# B&R Automation Studio project dbserv_0640 (part 4)

```c
/*=============================================================================
// Funktion: WorkEvent
//-----------------------------------------------------------------------------
// Zugriff auf das Prozessabbild.
// Input:	idBrServer: System-ID
// Return:	== 0 -> kein Fehler aufgetreten.
//			!= 0 -> Fehlerstatus der Funktion.
//=============================================================================*/

#ifdef FERTIG

UINT WorkEvent (void *idBrServer) {

	ACCESS_SERVER	*pAccessServer;
	ACCESS_UNIT		*pAccessUnit;
	ACCESS_TYPE		*pAccessType;
	ACCESS_POINT	*pAccessPoint;
	TYPE_DESC		*pTypeDesc;
	ITEM_DESC		*pItemDesc;

	ACCESS_ITEM_EVENT_LINK	*pAccessEventLinkItem;
	ACCESS_ITEM_EVENT_STATE	*pAccessEventItem;

	ACCESS_EVENT_PIPE	*pAccessEventPipe;
	EVENT_PIPE_HEADER	*pEventPipeHeader;
	EVENT_PIPE_DATA 	EventPipeData;
	USINT				*pEventPipeData, *pEventPipeTime;

	UDINT		lengthExtern, lengthPipeData, lengthTimeStamp;
	UINT		iPipeWrite, i;

	UINT		instance, unit, type, point, item;
	USINT		*pValue;
	UINT		lengthValue;
	USINT		eventtype;
	USINT		*pDataExtern;
	RTCtime_typ	RTCTime;

	if (idBrServer != NULL) {
		pAccessServer = (ACCESS_SERVER*)idBrServer;
		for (instance=0; instance<pAccessServer->countEventInstance; instance++) {
			for (unit=0; unit<pAccessServer->countUnit; unit++) {
				pAccessUnit = &pAccessServer->pAccessUnit[unit];
				if (pAccessUnit->pAccessType != NULL) {
					if (pAccessUnit->pUnitEventState[instance].countEvent > 0) {
						for (type=0; type<pAccessUnit->countType; type++) {
							pAccessType = &pAccessUnit->pAccessType[type];
							pTypeDesc = &pAccessServer->pAccessTypeDesc[type];
							if (pAccessType->pAccessPoint != NULL) {
								if (pAccessType->pTypeEventState[instance].countEvent > 0) {
									for (point=0; point<pAccessType->countPoint; point++) {
										pAccessPoint = &pAccessType->pAccessPoint[point];
										if (pAccessPoint->pAccessData != NULL) {
											if (pAccessPoint->pPointEventState[instance].countEvent > 0) {
												for (item=0; item<pTypeDesc->countItem ; item++) {
													pItemDesc = &pTypeDesc->pItemDesc[item];

													/* Event Datenbereich */
													pAccessEventItem = pAccessPoint->pAccessData + pAccessType->offiEvent + instance * pAccessType->leniEventNext + item * pAccessType->leniEventAlign;
													if (*pAccessEventItem == TRUE) {
														/* Link Datenbereich */
														pAccessEventLinkItem = pAccessPoint->pAccessData + pAccessType->offiEventlink + instance * pAccessType->leniEventlinkNext + item * pAccessType->leniEventlinkAlign;
														if (*pAccessEventLinkItem != cITEM_UNLINKED) {

															/* Daten wie für Funktions-Prototypen */
															pValue = pAccessPoint->pAccessData + pAccessType->offExtern + pItemDesc->offItem;
															lengthValue = pItemDesc->lenItem;
															eventtype = 0;
															pDataExtern = NULL;
															if (pAccessType->lenTime > 0) {
																memcpy(&RTCTime, pAccessPoint->pAccessData + pAccessType->offTime + item * pAccessType->lenTimeAlign, pAccessType->lenTime);
															}
															else {
																memset(&RTCTime, 0, sizeof(RTCTime));
															}

															/* SetEventItem */
															pAccessEventPipe = pAccessServer->pAccessEventPipe;
															lengthExtern = pItemDesc->lenItem;
															lengthTimeStamp = (*pAccessEventLinkItem == cITEM_LINKED_WITH_TIMESTAMP) ? sizeof(RTCtime_typ) : 0;
															pEventPipeHeader = (EVENT_PIPE_HEADER*)((USINT*)pAccessEventPipe[type].pEventPipeHeader + instance * pAccessEventPipe[type].length_pipe_next);
															lengthPipeData = (pValue != NULL) ? lengthValue : 0;
															if (pEventPipeHeader != NULL &&
																pEventPipeHeader->stateEvent.countEvent == 0 &&
																((pEventPipeHeader->iPipeWrite >= pEventPipeHeader->iPipeRead &&
																(UINT)(pEventPipeHeader->pipe_size - (pEventPipeHeader->iPipeWrite - pEventPipeHeader->iPipeRead)) > sizeof(EVENT_PIPE_DATA) + lengthTimeStamp + lengthPipeData) ||
																(pEventPipeHeader->iPipeWrite < pEventPipeHeader->iPipeRead &&
																(UINT)(pEventPipeHeader->iPipeRead - pEventPipeHeader->iPipeWrite) > sizeof(EVENT_PIPE_DATA) + lengthTimeStamp + lengthPipeData))) {

																if (pValue != NULL || pDataExtern != NULL) {
																	if ((pValue != NULL && lengthValue == lengthExtern) || pDataExtern != NULL) {
																		/* Eintrag in Event-Pipe */
																		iPipeWrite = pEventPipeHeader->iPipeWrite;

																		/* Header vorbesetzen */
																		EventPipeData.linkstate = *pAccessEventLinkItem;
																		EventPipeData.eventtype = eventtype;
																		EventPipeData.unit = unit;
																		EventPipeData.device = device;
																		EventPipeData.type = type;
																		EventPipeData.point= point;
																		EventPipeData.item = item;
																		EventPipeData.length = lengthValue;
																		EventPipeData.pData = pDataExtern;
																		pEventPipeData = (USINT*)&EventPipeData;
																		/* Header eintragen */
																		for (i=0; i<sizeof(EVENT_PIPE_DATA); i++) {
																			pEventPipeHeader->pPipeData[iPipeWrite++ % pEventPipeHeader->pipe_size] = pEventPipeData[i];
																		}
																		if (pValue != NULL) {
																			/* Daten eintragen */
																			for (i=0; i<lengthValue; i++) {
																				pEventPipeHeader->pPipeData[iPipeWrite++ % pEventPipeHeader->pipe_size] = pValue[i];
																			}
																		}
																		/* optional Zeitstempel eintragen */
																		if (lengthTimeStamp > 0) {
																			pEventPipeTime = (USINT*)&RTCTime;
																			for (i=0; i<lengthTimeStamp; i++) {
																				pEventPipeHeader->pPipeData[iPipeWrite++ % pEventPipeHeader->pipe_size] = pEventPipeTime[i];
																			}
																		}
																		/* Ereigniszeit aktualisieren */
																		if (pItemDesc->tsItem == TRUE) {
																			memcpy(pAccessPoint->pAccessData + pAccessType->offiTime + instance * pAccessType->leniTimeNext + item * pAccessType->leniTimeAlign, &RTCTime, pAccessType->leniTime);
																		}
																		pEventPipeHeader->iPipeWrite = (iPipeWrite % pEventPipeHeader->pipe_size); /* Index erst nach Zugriff updaten !!! */
																		pEventPipeHeader->pipe_level++; /* Füllstand erhöhen */

																	} /* ((pValue != NULL && lengthValue == lengthExtern) || pDataExtern != NULL) */
																	else {
																		return cEC_INVALID_LENGTH;
																	}
																} /* (pValue != NULL || pDataExtern != NULL) */
																else {
																	return cEC_INVALID_HANDLE;
																}
															}
														} /* (*pAccessEventLinkItem != cITEM_UNLINKED) */

														*pAccessEventItem = FALSE;
														pAccessPoint->pPointEventState[instance].countEvent--;
														pAccessType->pTypeEventState[instance].countEvent--;
														pAccessUnit->pUnitEventState[instance].countEvent--;

													} /* (*pAccessEventItem == TRUE) */
												} /* (item=0; item<pTypeDesc->countItem ; item++) */
											} /* (pAccessPoint->pPointEventState[instance] > 0) */
										} /* (pAccessPoint->pAccessData != NULL) */
									} /* (point=0; point<pAccessType->countPoint; point++) */
								} /* (pAccessType->pTypeEventState[instance].countEvent > 0) */
							} /* (pAccessType->pAccessPoint != NULL) */
						} /* (type=0; type<pAccessUnit->countType; type++) */
					} /* (pAccessUnit->pUnitEventState[instance].countEvent > 0) */
				} /* (pAccessUnit->pAccessType != NULL) */
			} /* (unit=0; unit<pAccessServer->countUnit; unit++) */
		} /* (instance=0; instance<pAccessServer->countEventInstance; instance++) */
		return cEC_OK;
	} /* (idBrServer != NULL) */
	else {
		return cEC_INVALID_SERVER;
	}
} /* WorkEvent */

/*UINT WorkEvent (void *idBrServer) {*/

	ACCESS_SERVER	*pAccessServer;
	ACCESS_UNIT		*pAccessUnit;
	ACCESS_TYPE		*pAccessType;
	ACCESS_POINT	*pAccessPoint;
	TYPE_DESC		*pTypeDesc;
	ITEM_DESC		*pItemDesc;
	ACCESS_ITEM_EVENT_LINK	*pAccessEventLinkItem;
	ACCESS_EVENT_PIPE		*pAccessEventPipe;
	EVENT_PIPE_HEADER		*pEventPipeHeader;

	UDINT					lengthExtern, lengthTimeStamp;
	UINT					i, instance, unit, device, type, point, iPipeWrite;

	EVENT_PIPE_DATA 		EventPipeData;
	USINT					*pEventPipeData, *pData, *pEventPipeTime;

	if (idBrServer != NULL) {
		pAccessServer = (ACCESS_SERVER*)idBrServer;
		for (instance=0; instance<pAccessServer->countEventInstance; instance++) {
			for (unit=0; unit<pAccessServer->countUnitNo; unit++) {
				pAccessUnit = &pAccessServer->pAccessUnit[unit];
				if (pAccessUnit->pAccessType != NULL) {
					if (pAccessServer->pUnitEventState[pAccessServer->countEventInstance * unit + instance].countEvent != 0) {
						for (device=0; device<pAccessUnit[unit].countDeviceNo; device++) {
							pAccessDevice = pAccessUnit[unit].pAccessDevice;
							if (device == pAccessDevice[device].device_no && pAccessDevice[device].pAccessType != NULL) {
								if (pAccessUnit[unit].pDeviceEventState[pAccessServer->countEventInstance * device + instance].countEvent != 0) {
									for (type=0; type<pAccessDevice[device].countType; type++) {
										if (pAccessDevice[device].pTypeEventState[pAccessServer->countEventInstance * type + instance].countEvent != 0) {

											pAccessType = pAccessDevice[device].pAccessType;
											pAccessEventPipe = pAccessServer->pAccessEventPipe;
											pEventPipeHeader = (EVENT_PIPE_HEADER*)((USINT*)pAccessEventPipe[type].pEventPipeHeader + instance * pAccessEventPipe[type].length_pipe_next);

											for (point=0; point<pAccessType[type].countPoint; point++) {

												pAccessEventLinkItem = pAccessType[type].pData_ieventlink + point * pAccessType[type].length_ieventlink_next;
												lengthExtern = pAccessEventPipe[type].TypeDefinition.length_extern;
												lengthTimeStamp = (pAccessEventLinkItem[instance] == cITEM_LINKED_WITH_TIMESTAMP) ? sizeof(RTCtime_typ) : 0;

												/* genügend Platz in der Event-Pipe ? */
												if (pEventPipeHeader != NULL &&
													pEventPipeHeader->stateEvent.countEvent != 0 &&
													((pEventPipeHeader->iPipeWrite >= pEventPipeHeader->iPipeRead &&
													(UINT)(pEventPipeHeader->pipe_size - (pEventPipeHeader->iPipeWrite - pEventPipeHeader->iPipeRead)) > sizeof(EVENT_PIPE_DATA) + lengthTimeStamp + lengthExtern) ||
													(pEventPipeHeader->iPipeWrite < pEventPipeHeader->iPipeRead &&
													(UINT)(pEventPipeHeader->iPipeRead - pEventPipeHeader->iPipeWrite) > sizeof(EVENT_PIPE_DATA) + lengthTimeStamp + lengthExtern))) {

													/* Event auf Datenpunkt vorhanden ? */
													if (*(UDINT*)(pAccessType[type].pData_ievent + point * pAccessType[type].length_ievent_next + instance * pAccessType[type].length_ievent_align) != 0 &&
														*(UDINT*)(pAccessType[type].pData_ievent + point * pAccessType[type].length_ievent_next + instance * pAccessType[type].length_ievent_align) == pEventPipeHeader->stateEvent.firstEvent) {

														/* Datenpunkt noch gelinkt ? */
														if (pAccessEventLinkItem[instance] != cITEM_UNLINKED) {

															/* Eintrag in Event-Pipe */
															iPipeWrite = pEventPipeHeader->iPipeWrite;

															/* Header eintragen */
															EventPipeData.linkstate = pAccessEventLinkItem[instance];
															EventPipeData.eventtype = 0;
															EventPipeData.unit = unit;
															EventPipeData.device = device;
															EventPipeData.type = type;
															EventPipeData.point= point;
															EventPipeData.item = 0;
															EventPipeData.length = lengthExtern;
															EventPipeData.pData = NULL;
															pEventPipeData = (USINT*)&EventPipeData;
															for (i=0; i<sizeof(EVENT_PIPE_DATA); i++) {
																pEventPipeHeader->pPipeData[iPipeWrite++ % pEventPipeHeader->pipe_size] = pEventPipeData[i];
															}

															/* Daten eintragen */
															pData = pAccessType[type].pData_extern + point * pAccessType[type].length_extern_align;
															for (i=0; i<lengthExtern; i++) {
																pEventPipeHeader->pPipeData[iPipeWrite++ % pEventPipeHeader->pipe_size] = pData[i];
															}
															pEventPipeHeader->iPipeWrite = (iPipeWrite % pEventPipeHeader->pipe_size); /* Index erst nach Zugriff updaten !!! */
															pEventPipeHeader->pipe_level++; /* Füllstand erhöhen */

															/* optional Zeitstempel eintragen */
															if (lengthTimeStamp > 0) {
																pEventPipeTime = pAccessType[type].pData_time + point * pAccessType[type].length_time_align;
																for (i=0; i<lengthTimeStamp; i++) {
																	pEventPipeHeader->pPipeData[iPipeWrite++ % pEventPipeHeader->pipe_size] = pEventPipeTime[i];
																}
															}
														} /* (pAccessItemLink[instance] != cITEM_UNLINKED) */

														/* Event auf Pipe-Typ austragen */
														pEventPipeHeader->stateEvent.firstEvent++;
														if (pEventPipeHeader->stateEvent.firstEvent > pEventPipeHeader->stateEvent.lastEvent) {
															pEventPipeHeader->stateEvent.firstEvent = 0;
															pEventPipeHeader->stateEvent.lastEvent = 0;
														}
														/* Event auf Punkt, Typ, Station, System austragen */
														*(UDINT*)(pAccessType[type].pData_ievent + point * pAccessType[type].length_ievent_next + instance * pAccessType[type].length_ievent_align) = 0;
														pEventPipeHeader->stateEvent.countEvent--;

														pAccessDevice[device].pTypeEventState[pAccessServer->countEventInstance * type + instance].countEvent--;
														pAccessUnit[unit].pDeviceEventState[pAccessServer->countEventInstance * device + instance].countEvent--;
														pAccessServer->pUnitEventState[pAccessServer->countEventInstance * unit + instance].countEvent--;

														/*if (pAccessServer->stateEvent[instance].countEvent == 0) {*/
															/* sicherheitshalber alle Pipe-Events bezüglich first/last austragen */
															/*for (m=0; m<pAccessServer->countType; m++) {
																pAccessEventPipe[m].stateEvent.firstEvent = 0;
																pAccessEventPipe[m].stateEvent.lastEvent = 0;
															}*/
														/*} (pAccessSystem->stateEvent.countEvent == 0) */
													} /* ... */
												} /* ... */
												else {
													break;
												}
											} /* (point=0; point<pAccessType[type].countPoint; point++) */
										} /* (pAccessDevice[device].pTypeEventState[pAccessServer->countEventInstance * type + instance].countEvent != 0) */
									} /* (type=0; type<pAccessDevice[device].countType; type++) */
								} /* (pAccessUnit[unit].pDeviceEventState[pAccessServer->countEventInstance * device + instance].countEvent != 0) */
							} /* (device == pAccessDevice[device].device_no && pAccessDevice[device].pAccessType != NULL) */
						} /* (device=0; device<pAccessUnit.countDeviceNo; device++) */
					} /* (pAccessServer->pUnitEventState[pAccessServer->countInstance * unit + instance].countEvent != 0) */
				} /* (unit == pAccessUnit[unit].unit_no && pAccessUnit[unit].pAccessDevice != NULL) */
			} /* (unit=0; unit<pAccessServer->countUnitNo; unit++) */
		} /* (instance=0; instance<pAccessServer->countEventInstance; instance++) */
		return cEC_OK;
	} /* (idBrServer != NULL) */
	else {
		return cEC_INVALID_SERVER;
	}
} /* work_event */
#endif

/*=============================================================================
// Funktion: LinkWriteInstance
//-----------------------------------------------------------------------------
// System mit allen zugehörigen Datenpunkten für die Ereignisbehandlung anmelden.
// Input:	idBrServer: System-ID
//			instance:	Instanz-Nummer
// Return:	== 0 -> kein Fehler aufgetreten.
//			!= 0 -> Fehlerstatus der Funktion.
//=============================================================================*/

UINT LinkWriteInstance (void *idBrServer, UINT instance) {

	ACCESS_SERVER	*pAccessServer;
	ACCESS_UNIT		*pAccessUnit;
	ACCESS_TYPE		*pAccessType;
	ACCESS_POINT	*pAccessPoint;
	TYPE_DESC		*pTypeDesc;
	ACCESS_ITEM_WRITE_LINK	*pAccessWriteLinkItem;

	unsigned short	unit, type, point, item;

	if (idBrServer != NULL) {
		pAccessServer = (ACCESS_SERVER*)idBrServer;
		if (instance < pAccessServer->countWriteInstance) {
			for (unit=0; unit<pAccessServer->countUnit; unit++) {
				pAccessUnit = &pAccessServer->pAccessUnit[unit];
				if (pAccessUnit->pAccessType != NULL) {
					for (type=0; type<pAccessUnit->countType; type++) {
						pAccessType = &pAccessUnit->pAccessType[type];
						pTypeDesc = &pAccessServer->pAccessTypeDesc[type];
						if (pAccessType->pAccessPoint != NULL) {
							for (point=0; point<pAccessType->countPoint; point++) {
								pAccessPoint = &pAccessType->pAccessPoint[point];
								if (pAccessPoint->pAccessData != NULL) {
									for (item=0; item<pTypeDesc->countItem ; item++) {
										/* Link Datenbereich */
										pAccessWriteLinkItem = pAccessPoint->pAccessData + pAccessType->offWritelink + item * pAccessType->lenWritelinkAlign;
										if (*pAccessWriteLinkItem == 0) {
											*pAccessWriteLinkItem = instance + 1;
										}
									} /* (item = 0; item<pTypeDesc->countItem ; item++) */
								} /* (pAccessPoint->pAccessData != NULL) */
							} /* (point=0; point<pAccessType->countPoint; point++) */
						} /* (pAccessType->pAccessPoint != NULL) */
					} /* (type=0; type<pAccessUnit->countType; type++) */
				} /* (pAccessUnit->pAccessType != NULL) */
			} /* (unit=0; unit<pAccessServer->countUnit; unit++) */
			return cEC_OK;
		} /* (instance < pAccessSystem->countWriteInstance) */
		else {
			return cEC_INVALID_INSTANCE;
		}
	} /* (idBrServer != NULL) */
	else {
		return cEC_INVALID_SERVER;
	}
} /* LinkWriteInstance */

/*=============================================================================
// Funktion: UnlinkWriteInstance
//-----------------------------------------------------------------------------
// System mit allen zugehörigen Datenpunkten für die Ereignisbehandlung anmelden.
// Input:	idBrServer: System-ID
//			instance:	Instanz-Nummer
// Return:	== 0 -> kein Fehler aufgetreten.
//			!= 0 -> Fehlerstatus der Funktion.
//=============================================================================*/

UINT UnlinkWriteInstance (void *idBrServer, UINT instance) {

	ACCESS_SERVER	*pAccessServer;
	ACCESS_UNIT		*pAccessUnit;
	ACCESS_TYPE		*pAccessType;
	ACCESS_POINT	*pAccessPoint;
	TYPE_DESC		*pTypeDesc;
	ACCESS_ITEM_WRITE_LINK	*pAccessWriteLinkItem;

	unsigned short	unit, type, point, item;

	if (idBrServer != NULL) {
		pAccessServer = (ACCESS_SERVER*)idBrServer;
		if (instance < pAccessServer->countWriteInstance) {
			for (unit=0; unit<pAccessServer->countUnit; unit++) {
				pAccessUnit = &pAccessServer->pAccessUnit[unit];
				if (pAccessUnit->pAccessType != NULL) {
					for (type=0; type<pAccessUnit->countType; type++) {
						pAccessType = &pAccessUnit->pAccessType[type];
						pTypeDesc = &pAccessServer->pAccessTypeDesc[type];
						if (pAccessType->pAccessPoint != NULL) {
							for (point=0; point<pAccessType->countPoint; point++) {
								pAccessPoint = &pAccessType->pAccessPoint[point];
								if (pAccessPoint->pAccessData != NULL) {
									for (item=0; item<pTypeDesc->countItem ; item++) {
										/* Unlink Datenbereich */
										pAccessWriteLinkItem = pAccessPoint->pAccessData + pAccessType->offWritelink + item * pAccessType->lenWritelinkAlign;
										if (*pAccessWriteLinkItem > 0) {
											*pAccessWriteLinkItem = 0;
										}
									} /* (item = 0; item<pTypeDesc->countItem ; item++) */
								} /* (pAccessPoint->pAccessData != NULL) */
							} /* (point=0; point<pAccessType->countPoint; point++) */
						} /* (pAccessType->pAccessPoint != NULL) */
					} /* (type=0; type<pAccessUnit->countType; type++) */
				} /* (pAccessUnit->pAccessType != NULL) */
			} /* (unit=0; unit<pAccessServer->countUnit; unit++) */
			return cEC_OK;
		} /* (instance < pAccessSystem->countWriteInstance) */
		else {
			return cEC_INVALID_INSTANCE;
		}
	} /* (idBrServer != NULL) */
	else {
		return cEC_INVALID_SERVER;
	}
} /* UnlinkWriteInstance */

/*=============================================================================
// Funktion: LinkWriteItem
//-----------------------------------------------------------------------------
// Datenpunkt für Ereignisbehandlung anmelden.
// Input:	idBrServer: System-ID
//			instance:	Instanz-Nummer
//			unit:		Anlagen-Nummer
//			device:		Gerät-Nummer
//			type:		Datentyp-Nummer
//			point:		Datenpunkt-Nummer
//			item:		Strukturelement-Nummer
// Return:	== 0 -> kein Fehler aufgetreten.
//			!= 0 -> Fehlerstatus der Funktion.
//=============================================================================*/

UINT LinkWriteItem (void *idBrServer, UINT instance,
					UINT unit, UINT device, UINT type, UINT point, UINT item,
					UDINT handle) {

	ACCESS_SERVER	*pAccessServer;
	ACCESS_UNIT		*pAccessUnit;
	ACCESS_TYPE		*pAccessType;
	ACCESS_POINT	*pAccessPoint;
	TYPE_DESC		*pTypeDesc;
	ITEM_DESC		*pItemDesc;
	ACCESS_ITEM_WRITE_LINK		*pAccessWriteLinkItem;
	ACCESS_ITEM_WRITE_HANDLE	*pAccessWriteHandleItem;

	if (idBrServer != NULL) {
		pAccessServer = (ACCESS_SERVER*)idBrServer;
		if (instance < pAccessServer->countWriteInstance) {
			if (unit < pAccessServer->countUnit && pAccessServer->pAccessUnit[unit].pAccessType != NULL) {
				pAccessUnit = &pAccessServer->pAccessUnit[unit];
				if (device == pAccessServer->noDevice) {
					if (type < pAccessUnit->countType && pAccessUnit->pAccessType[type].pAccessPoint != NULL) {
						pAccessType = &pAccessUnit->pAccessType[type];
						pTypeDesc = &pAccessServer->pAccessTypeDesc[type];
						if (point < pAccessType->countPoint && pAccessType->pAccessPoint[point].pAccessData != NULL) {
							pAccessPoint = &pAccessType->pAccessPoint[point];
							if (item < pTypeDesc->countItem) {
								pItemDesc = &pTypeDesc->pItemDesc[item];

								/* Link Datenbereich */
								pAccessWriteLinkItem = pAccessPoint->pAccessData + pAccessType->offWritelink + item * pAccessType->lenWritelinkAlign;
								pAccessWriteHandleItem = (ACCESS_ITEM_WRITE_HANDLE*)(pAccessPoint->pAccessData + pAccessType->offWritehandle + item * pAccessType->lenWritehandleAlign);
								if (*pAccessWriteLinkItem == 0) {
									*pAccessWriteLinkItem = instance + 1;
									*pAccessWriteHandleItem = handle;
									return cEC_OK;
								}
								else {
									return cEC_ITEM_ALREADY_LINKED;
								}

							} /* (item < pTypeDesc->countItem) */
							else {
								return cEC_INVALID_ITEM;
							}
						} /* (point < pAccessType->countPoint && pAccessType->pAccessPoint[point].pAccessData != NULL) */
						else {
							return cEC_INVALID_POINT;
						}
					} /* (type < pAccessUnit->countType && pAccessUnit->pAccessType[type].pAccessPoint != NULL) */
					else {
						return cEC_INVALID_TYPE;
					}
				} /* (device == pAccessServer->noDevice) */
				else {
					return cEC_INVALID_DEVICE;
				}
			} /* (unit < pAccessServer->countUnit) */
			else {
				return cEC_INVALID_UNIT;
			}
		} /* (instance < pAccessSystem->countWriteInstance) */
		else {
			return cEC_INVALID_INSTANCE;
		}
	} /* (idBrServer != NULL) */
	else {
		return cEC_INVALID_SERVER;
	}
} /* LinkWriteItem */

/*=============================================================================
// Funktion: UnlinkWriteItem
//-----------------------------------------------------------------------------
// Datenpunkt für Ereignisbehnadlung abmelden.
// Input:	idBrServer: System-ID
//			instance:	Instanz-Nummer
//			unit:		Anlagen-Nummer
//			device:		Gerät-Nummer
//			type:		Datentyp-Nummer
//			point:		Datenpunkt-Nummer
//			item:		Strukturelement-Nummer
// Return:	== 0 -> kein Fehler aufgetreten.
//			!= 0 -> Fehlerstatus der Funktion.
//=============================================================================*/

UINT UnlinkWriteItem (void *idBrServer, UINT instance,
						UINT unit, UINT device, UINT type, UINT point, UINT item) {

	ACCESS_SERVER	*pAccessServer;
	ACCESS_UNIT		*pAccessUnit;
	ACCESS_TYPE		*pAccessType;
	ACCESS_POINT	*pAccessPoint;
	TYPE_DESC		*pTypeDesc;
	ITEM_DESC		*pItemDesc;
	ACCESS_ITEM_WRITE_LINK		*pAccessWriteLinkItem;
	ACCESS_ITEM_WRITE_HANDLE	*pAccessWriteHandleItem;

	if (idBrServer != NULL) {
		pAccessServer = (ACCESS_SERVER*)idBrServer;
		if (instance < pAccessServer->countWriteInstance) {
			if (unit < pAccessServer->countUnit && pAccessServer->pAccessUnit[unit].pAccessType != NULL) {
				pAccessUnit = &pAccessServer->pAccessUnit[unit];
				if (device == pAccessServer->noDevice) {
					if (type < pAccessUnit->countType && pAccessUnit->pAccessType[type].pAccessPoint != NULL) {
						pAccessType = &pAccessUnit->pAccessType[type];
						pTypeDesc = &pAccessServer->pAccessTypeDesc[type];
						if (point < pAccessType->countPoint && pAccessType->pAccessPoint[point].pAccessData != NULL) {
							pAccessPoint = &pAccessType->pAccessPoint[point];
							if (item < pTypeDesc->countItem) {
								pItemDesc = &pTypeDesc->pItemDesc[item];

								/* Unlink Datenbereich */
								pAccessWriteLinkItem = pAccessPoint->pAccessData + pAccessType->offWritelink + item * pAccessType->lenWritelinkAlign;
								pAccessWriteHandleItem = (ACCESS_ITEM_WRITE_HANDLE*)(pAccessPoint->pAccessData + pAccessType->offWritehandle + item * pAccessType->lenWritehandleAlign);
								if (*pAccessWriteLinkItem > 0) {
									*pAccessWriteLinkItem = 0;
									*pAccessWriteHandleItem = 0;
									return cEC_OK;
								}
								else {
									return cEC_ITEM_ALREADY_UNLINKED;
								}

							} /* (item < pTypeDesc->countItem) */
							else {
								return cEC_INVALID_ITEM;
							}
						} /* (point < pAccessType->countPoint && pAccessType->pAccessPoint[point].pAccessData != NULL) */
						else {
							return cEC_INVALID_POINT;
						}
					} /* (type < pAccessUnit->countType && pAccessUnit->pAccessType[type].pAccessPoint != NULL) */
					else {
						return cEC_INVALID_TYPE;
					}
				} /* (device == pAccessServer->noDevice) */
				else {
					return cEC_INVALID_DEVICE;
				}
			} /* (unit < pAccessServer->countUnit && pAccessServer->pAccessUnit[unit].pAccessType != NULL) */
			else {
				return cEC_INVALID_UNIT;
			}
		} /* (instance < pAccessSystem->countWriteInstance) */
		else {
			return cEC_INVALID_INSTANCE;
		}
	} /* (idBrServer != NULL) */
	else {
		return cEC_INVALID_SERVER;
	}
} /* UnlinkWriteItem */

/*=============================================================================
// Funktion: SetWriteItem
//-----------------------------------------------------------------------------
// Zugriff auf das Prozessabbild.
// Input:	idBrServer: System-ID
//			system:		Anlagen-Nummer
//			station:	Stations-Nummer
//			type:		Datentyp-Nummer
//			point:		Datenpunkt-Nummer
//			ppData_extern:	Zeiger auf externen Datenbereich (Rückgabewert)
//			plength_extern:	Länge des externen Datenbereichs (Rückgabewert)
//			ppData_intern:	Zeiger auf internen Datenbereich (Rückgabewert)
//			plength_intern:	Länge des internen Datenbereichs (Rückgabewert)
//			ppData_time:	Zeiger auf Zeitbereich (Rückgabewert)
//			plength_time:	Länge des Zeitbereichs (Rückgabewert)
//			ppData_event:	Zeiger auf Ereignis-Kennung (Rückgabewert)
//			plength_event:	Länge der Ereignis-Kennung (Rückgabewert)
// Return:	== 0 -> kein Fehler aufgetreten.
//			!= 0 -> Fehlerstatus der Funktion.
//=============================================================================*/

UINT SetWriteItem (void *idBrServer,
					UINT unit, UINT device, UINT type, UINT point, UINT item,
					USINT* pValue, UDINT lengthValue) {

	ACCESS_SERVER	*pAccessServer;
	ACCESS_UNIT		*pAccessUnit;
	ACCESS_TYPE		*pAccessType;
	ACCESS_POINT	*pAccessPoint;
	TYPE_DESC		*pTypeDesc;
	ITEM_DESC		*pItemDesc;
	ACCESS_WRITE_PIPE			*pAccessWritePipe;
	WRITE_PIPE_HEADER			*pWritePipeHeader;
	ACCESS_ITEM_WRITE_LINK		*pAccessWriteLinkItem;
	ACCESS_ITEM_WRITE_HANDLE	*pAccessWriteHandleItem;

	UDINT			lengthExtern;
	UINT			instance, iPipeWrite, i;

	WRITE_PIPE_DATA	WritePipeData;
	USINT			*pWritePipeData;

	if (idBrServer != NULL) {
		pAccessServer = (ACCESS_SERVER*)idBrServer;
		if (unit < pAccessServer->countUnit && pAccessServer->pAccessUnit[unit].pAccessType != NULL) {
			pAccessUnit = &pAccessServer->pAccessUnit[unit];
			if (device == pAccessServer->noDevice) {
				if (type < pAccessUnit->countType && pAccessUnit->pAccessType[type].pAccessPoint != NULL) {
					pAccessType = &pAccessUnit->pAccessType[type];
					pTypeDesc = &pAccessServer->pAccessTypeDesc[type];
					if (point < pAccessType->countPoint && pAccessType->pAccessPoint[point].pAccessData != NULL) {
						pAccessPoint = &pAccessType->pAccessPoint[point];
						if (item < pTypeDesc->countItem) {
							pItemDesc = &pTypeDesc->pItemDesc[item];
							pAccessWriteLinkItem = pAccessPoint->pAccessData + pAccessType->offWritelink + item * pAccessType->lenWritelinkAlign;
							pAccessWriteHandleItem = (ACCESS_ITEM_WRITE_HANDLE*)(pAccessPoint->pAccessData + pAccessType->offWritehandle + item * pAccessType->lenWritehandleAlign);
							if (*pAccessWriteLinkItem > 0) {
								instance = *pAccessWriteLinkItem - 1;
								pAccessWritePipe = pAccessServer->pAccessWritePipe;
								lengthExtern = pItemDesc->lenItem;
								pWritePipeHeader = (WRITE_PIPE_HEADER*)((USINT*)pAccessWritePipe->pWritePipeHeader + instance * pAccessWritePipe->length_pipe_next);
								if (pWritePipeHeader != NULL
									&&
									(
										(
											pWritePipeHeader->iPipeWrite >= pWritePipeHeader->iPipeRead &&
											(UINT)(pWritePipeHeader->pipe_size - (pWritePipeHeader->iPipeWrite - pWritePipeHeader->iPipeRead)) > sizeof(WRITE_PIPE_DATA) + lengthValue
										)
										||
										(
											pWritePipeHeader->iPipeWrite < pWritePipeHeader->iPipeRead &&
											(UINT)(pWritePipeHeader->iPipeRead - pWritePipeHeader->iPipeWrite) > sizeof(WRITE_PIPE_DATA) + lengthValue
										)
									)
								) {
									if (pValue != NULL) {
										if (lengthValue == lengthExtern) {
											/* Eintrag in Event-Pipe */
											iPipeWrite = pWritePipeHeader->iPipeWrite;

											/* Header eintragen */
											WritePipeData.linkstate = cITEM_LINKED_WITHOUT_TIMESTAMP;
											WritePipeData.eventtype = 0;
											WritePipeData.unit = unit;
											WritePipeData.device = device;
											WritePipeData.type = type;
											WritePipeData.point= point;
											WritePipeData.item = item;
											WritePipeData.length = lengthValue;
											WritePipeData.pData = (USINT*)*pAccessWriteHandleItem;
											pWritePipeData = (USINT*)&WritePipeData;
											/* Header eintragen */
											for (i=0; i<sizeof(WRITE_PIPE_DATA); i++) {
												pWritePipeHeader->pPipeData[iPipeWrite++ % pWritePipeHeader->pipe_size] = pWritePipeData[i];
											}
											if (pValue != NULL) {
												/* Daten eintragen */
												for (i=0; i<lengthValue; i++) {
													pWritePipeHeader->pPipeData[iPipeWrite++ % pWritePipeHeader->pipe_size] = pValue[i];
												}
											}
											pWritePipeHeader->iPipeWrite = (iPipeWrite % pWritePipeHeader->pipe_size); /* Index erst nach Zugriff updaten !!! */
											pWritePipeHeader->pipe_level++; /* Füllstand erhöhen */
											return cEC_OK;
										} /* (lengthValue == lengthExtern) */
										else {
											return cEC_INVALID_LENGTH;
										}
									} /* (pValue != NULL) */
									else {
										return cEC_INVALID_HANDLE;
									}
								} /* ... */
								else {
									return cEC_WRITE_PIPE_FULL;
								}
							} /* (*pAccessWriteLinkItem > 0) */
							else {
								return cEC_ITEM_NOT_WRITEABLE;
							}
						} /* (item < pTypeDesc->countItem) */
						else {
							return cEC_INVALID_ITEM;
						}
					} /* (point < pAccessType->countPoint && pAccessType->pAccessPoint[point].pAccessData != NULL) */
					else {
						return cEC_INVALID_POINT;
					}
				} /* (type < pAccessUnit->countType && pAccessUnit->pAccessType[type].pAccessPoint != NULL) */
				else {
					return cEC_INVALID_TYPE;
				}
			} /* (device == pAccessServer->noDevice) */
			else {
				return cEC_INVALID_DEVICE;
			}
		} /* (unit < pAccessServer->countUnitNo) */
		else {
			return cEC_INVALID_UNIT;
		}
	} /* (idBrServer != NULL) */
	else {
		return cEC_INVALID_SERVER;
	}
} /* SetWriteItem */

/*=============================================================================
// Funktion: ScanWriteItem
//-----------------------------------------------------------------------------
// Zugriff auf das Prozessabbild.
// Input:	idBrServer: System-ID
//			system:		Anlagen-Nummer
//			station:	Stations-Nummer
//			type:		Datentyp-Nummer
//			point:		Datenpunkt-Nummer
//			ppData_extern:	Zeiger auf externen Datenbereich (Rückgabewert)
//			plength_extern:	Länge des externen Datenbereichs (Rückgabewert)
//			ppData_intern:	Zeiger auf internen Datenbereich (Rückgabewert)
//			plength_intern:	Länge des internen Datenbereichs (Rückgabewert)
//			ppData_time:	Zeiger auf Zeitbereich (Rückgabewert)
//			plength_time:	Länge des Zeitbereichs (Rückgabewert)
//			ppData_event:	Zeiger auf Ereignis-Kennung (Rückgabewert)
//			plength_event:	Länge der Ereignis-Kennung (Rückgabewert)
// Return:	== 0 -> kein Fehler aufgetreten.
//			!= 0 -> Fehlerstatus der Funktion.
//=============================================================================*/

UINT ScanWriteItem (void *idBrServer, UINT instance,
					USINT* pWriteBuffer, UDINT lengthWriteBuffer,
					UDINT* pLength, UDINT* pLengthTimeStamp) {

	ACCESS_SERVER		*pAccessServer;
	ACCESS_WRITE_PIPE	*pAccessWritePipe;
	WRITE_PIPE_HEADER	*pWritePipeHeader;

	UINT				i, iPipeRead;
	UDINT				lengthExtern, lengthTimeStamp;

	WRITE_PIPE_DATA 	WritePipeData;
	USINT				*pWritePipeData;

	if (idBrServer != NULL) {
		pAccessServer = (ACCESS_SERVER*)idBrServer;
		if (instance < pAccessServer->countWriteInstance) {

			pAccessWritePipe = pAccessServer->pAccessWritePipe;
			pWritePipeHeader = (WRITE_PIPE_HEADER*)((USINT*)pAccessWritePipe->pWritePipeHeader + instance * pAccessWritePipe->length_pipe_next);
			if (pWritePipeHeader != NULL) {
				while (pWritePipeHeader->iPipeRead != pWritePipeHeader->iPipeWrite) {
					/* Eintrag in Event-Pipe */
					iPipeRead = pWritePipeHeader->iPipeRead;
					/* Header kopieren */
					pWritePipeData = (USINT*)&WritePipeData;
					for (i=0; i<sizeof(WRITE_PIPE_DATA); i++) {
						pWritePipeData[i] = pWritePipeHeader->pPipeData[iPipeRead++ % pWritePipeHeader->pipe_size];
					}
					lengthExtern = WritePipeData.length;
					lengthTimeStamp = (WritePipeData.linkstate == cITEM_LINKED_WITH_TIMESTAMP) ? sizeof(RTCtime_typ) : 0;
					if (WritePipeData.linkstate == cITEM_UNLINKED) {
						iPipeRead = iPipeRead + lengthExtern + lengthTimeStamp;
						pWritePipeHeader->iPipeRead = (iPipeRead % pWritePipeHeader->pipe_size); /* Index erst nach Zugriff updaten !!! */
						pWritePipeHeader->pipe_level--; /* Füllstand vermindern */
						continue;
					}
					if (pLength != NULL) {
						*pLength = lengthExtern;
					}
					if (pLengthTimeStamp != NULL) {
						*pLengthTimeStamp = lengthTimeStamp;
					}
					/* Buffergröße überprüfen */
					if (sizeof(WRITE_PIPE_DATA) + lengthExtern + lengthTimeStamp <= lengthWriteBuffer) {
						/* Header austragen */
						for (i=0; i<sizeof(WRITE_PIPE_DATA); i++) {
							pWriteBuffer[i] = pWritePipeData[i];
						}
						/* Daten austragen */
						for (i=0; i<lengthExtern + lengthTimeStamp; i++) {
							pWriteBuffer[i + sizeof(WRITE_PIPE_DATA)] = pWritePipeHeader->pPipeData[iPipeRead++ % pWritePipeHeader->pipe_size];
						}
						return cEC_OK;
					}
					else {
						return cEC_EVENTBUFFER_TO_SMALL;
					}
				} /* (pEventPipeHeader->iPipeRead != pEventPipeHeader->iPipeWrite) */
			} /* (pWritePipeHeader != NULL) */
			return cEC_NO_DATA_IN_WRITEBUFFER;
		} /* (instance < pAccessSystem->countWriteInstance) */
		else {
			return cEC_INVALID_INSTANCE;
		}
	} /* (idBrServer != NULL) */
	else {
		return cEC_INVALID_SERVER;
	}
} /* ScanWriteItem */

/*=============================================================================
// Funktion: GetWriteItem
//-----------------------------------------------------------------------------
// Zugriff auf das Prozessabbild.
// Input:	idBrServer: System-ID
//			system:		Anlagen-Nummer
//			station:	Stations-Nummer
//			type:		Datentyp-Nummer
//			point:		Datenpunkt-Nummer
//			ppData_extern:	Zeiger auf externen Datenbereich (Rückgabewert)
//			plength_extern:	Länge des externen Datenbereichs (Rückgabewert)
//			ppData_intern:	Zeiger auf internen Datenbereich (Rückgabewert)
//			plength_intern:	Länge des internen Datenbereichs (Rückgabewert)
//			ppData_time:	Zeiger auf Zeitbereich (Rückgabewert)
//			plength_time:	Länge des Zeitbereichs (Rückgabewert)
//			ppData_event:	Zeiger auf Ereignis-Kennung (Rückgabewert)
//			plength_event:	Länge der Ereignis-Kennung (Rückgabewert)
// Return:	== 0 -> kein Fehler aufgetreten.
//			!= 0 -> Fehlerstatus der Funktion.
//=============================================================================*/

UINT GetWriteItem (void *idBrServer, UINT instance,
					USINT* pWriteBuffer, UDINT lengthWriteBuffer,
					UDINT* pLength, UDINT* pLengthTimeStamp) {

	ACCESS_SERVER		*pAccessServer;
	ACCESS_WRITE_PIPE	*pAccessWritePipe;
	WRITE_PIPE_HEADER	*pWritePipeHeader;

	UINT				i, iPipeRead;
	UDINT				lengthExtern, lengthTimeStamp;

	WRITE_PIPE_DATA 	WritePipeData;
	USINT				*pWritePipeData;

	if (idBrServer != NULL) {
		pAccessServer = (ACCESS_SERVER*)idBrServer;
		if (instance < pAccessServer->countWriteInstance) {

			pAccessWritePipe = pAccessServer->pAccessWritePipe;
			pWritePipeHeader = (WRITE_PIPE_HEADER*)((USINT*)pAccessWritePipe->pWritePipeHeader + instance * pAccessWritePipe->length_pipe_next);
			if (pWritePipeHeader != NULL) {
				while (pWritePipeHeader->iPipeRead != pWritePipeHeader->iPipeWrite) {
					/* Eintrag in Event-Pipe */
					iPipeRead = pWritePipeHeader->iPipeRead;
					/* Header kopieren */
					pWritePipeData = (USINT*)&WritePipeData;
					for (i=0; i<sizeof(WRITE_PIPE_DATA); i++) {
						pWritePipeData[i] = pWritePipeHeader->pPipeData[iPipeRead++ % pWritePipeHeader->pipe_size];
					}
					lengthExtern = WritePipeData.length;
					lengthTimeStamp = (WritePipeData.linkstate == cITEM_LINKED_WITH_TIMESTAMP) ? sizeof(RTCtime_typ) : 0;
					if (WritePipeData.linkstate == cITEM_UNLINKED) {
						iPipeRead = iPipeRead + lengthExtern + lengthTimeStamp;
						pWritePipeHeader->iPipeRead = (iPipeRead % pWritePipeHeader->pipe_size); /* Index erst nach Zugriff updaten !!! */
						pWritePipeHeader->pipe_level--; /* Füllstand vermindern */
						continue;
					}
					if (pLength != NULL) {
						*pLength = lengthExtern;
					}
					if (pLengthTimeStamp != NULL) {
						*pLengthTimeStamp = lengthTimeStamp;
					}
					/* Buffergröße überprüfen */
					if (sizeof(WRITE_PIPE_DATA) + lengthExtern + lengthTimeStamp <= lengthWriteBuffer) {
						/* Header austragen */
						for (i=0; i<sizeof(WRITE_PIPE_DATA); i++) {
							pWriteBuffer[i] = pWritePipeData[i];
						}
						/* Daten austragen */
						for (i=0; i<lengthExtern + lengthTimeStamp; i++) {
							pWriteBuffer[i + sizeof(WRITE_PIPE_DATA)] = pWritePipeHeader->pPipeData[iPipeRead++ % pWritePipeHeader->pipe_size];
						}
						pWritePipeHeader->iPipeRead = (iPipeRead % pWritePipeHeader->pipe_size); /* Index erst nach Zugriff updaten !!! */
						pWritePipeHeader->pipe_level--; /* Füllstand vermindern */
						return cEC_OK;
					}
					else {
						return cEC_EVENTBUFFER_TO_SMALL;
					}
				} /* (pEventPipeHeader->iPipeRead != pEventPipeHeader->iPipeWrite) */
			} /* (pWritePipeHeader != NULL) */
			return cEC_NO_DATA_IN_WRITEBUFFER;
		} /* (instance < pAccessSystem->countWriteInstance) */
		else {
			return cEC_INVALID_INSTANCE;
		}
	} /* (idBrServer != NULL) */
	else {
		return cEC_INVALID_SERVER;
	}
} /* GetWriteItem */

/*=============================================================================
// Funktion: CopyPipeToFile
//-----------------------------------------------------------------------------
// Zugriff auf das Prozessabbild.
// Input:	idBrServer: System-ID
//			system:		Anlagen-Nummer
//			station:	Stations-Nummer
//			type:		Datentyp-Nummer
//			point:		Datenpunkt-Nummer
//			ppData_extern:	Zeiger auf externen Datenbereich (Rückgabewert)
//			plength_extern:	Länge des externen Datenbereichs (Rückgabewert)
//			ppData_intern:	Zeiger auf internen Datenbereich (Rückgabewert)
//			plength_intern:	Länge des internen Datenbereichs (Rückgabewert)
//			ppData_time:	Zeiger auf Zeitbereich (Rückgabewert)
//			plength_time:	Länge des Zeitbereichs (Rückgabewert)
//			ppData_event:	Zeiger auf Ereignis-Kennung (Rückgabewert)
//			plength_event:	Länge der Ereignis-Kennung (Rückgabewert)
// Return:	== 0 -> kein Fehler aufgetreten.
//			!= 0 -> Fehlerstatus der Funktion.
//=============================================================================*/

/*
	ltoa  converts a signed long  value into ASCII Format
	ultoa converts a unsigned long  value into ASCII Format

	both returns the length of the converted string.
*/

int ultoa(unsigned long value, char *buffer) {

	int string_len=0, i, j;
	char swap;

	do {
		buffer[string_len++]=(value % 10) + '0'; /*calculate next digit*/
	} while((value = value/10)); /*while there are more digits*/

	/*swap digits*/
	i=0;
	j=string_len-1;

	while (i<j) {
		swap = buffer[i];
		buffer[i] = buffer[j];
		buffer[j] = swap;
		i++; j--;
	}
	buffer[string_len]=0; /*NULL termination of string*/
	return string_len;    /*Return lenght of string*/
}

int ltoa(long value, char *buffer) {

	int string_len=0, neg=0, i, j;
	char swap;
	unsigned long absval;  /*we have to use unsigned long because, with signed long
	                         0x80000000 would not work.*/

	if (value<0) {
		absval = -value;
		neg=1;
		buffer[0]='-';
		string_len=1;
	}
	else {
		absval = value;
	}
	do {
		buffer[string_len++]=(absval % 10) + '0'; /*calculate next digit*/
	} while((absval = absval/10)); /*while there are more digits*/

	/*swap digits*/
	i=neg;  /*begin at pos 1 if negative*/
	j=string_len-1;

	while (i<j) {
		swap = buffer[i];
		buffer[i] = buffer[j];
		buffer[j] = swap;
		i++; j--;
	}
	buffer[string_len]=0; /*NULL termination of string*/
	return string_len;    /*Return lenght of string*/
}

UINT CopyPipeToFile (void *idBrServer) {

	ACCESS_SERVER		*pAccessServer;
	ACCESS_EVENT_PIPE	*pAccessEventPipe;
	EVENT_PIPE_INSTANCE	*pEventPipeInstance;
	EVENT_PIPE_HEADER	*pEventPipeHeaderWrite, *pEventPipeHeaderRead;
	UINT				instance, type;

	if (idBrServer != NULL) {
		pAccessServer = (ACCESS_SERVER*)idBrServer;
		for (instance = 0; instance < pAccessServer->countEventInstance; instance++) {
			for (type = 0; type < pAccessServer->countType; type++) {
				pAccessEventPipe = &pAccessServer->pAccessEventPipe[type];
				if (pAccessEventPipe->pEventPipeInstance != NULL) {
					pEventPipeInstance = &pAccessEventPipe->pEventPipeInstance[instance];
					#warning WriteToFile
					if (pAccessEventPipe->WriteToFile == TRUE) {

						pEventPipeHeaderWrite = pEventPipeInstance->pEventPipeHeaderWrite[pEventPipeInstance->BufferFileIndex];
						pEventPipeHeaderRead  = pEventPipeInstance->pEventPipeHeaderRead;

						if (pEventPipeHeaderWrite != NULL && pEventPipeHeaderRead != NULL) {

							/* ---------------- */
							/* File - Schreiben */
							/* ---------------- */
							switch (pEventPipeInstance->fileStep) {

								/* ------- */
								/* default */
								/* ------- */
								case 0:
									if (pEventPipeInstance->BufferEventIndex != pEventPipeInstance->BufferFileIndex)
									{
										if (1==0 && pEventPipeHeaderRead->iPipeWrite == pEventPipeHeaderRead->iPipeRead) {
										}
										else {
											pEventPipeInstance->fileState = 65535;

											pEventPipeInstance->WriteDataBusy = TRUE;
											pEventPipeInstance->ReadDataBusy = TRUE;

											pEventPipeInstance->WriteDataBusy = FALSE;
											pEventPipeInstance->ReadDataBusy = FALSE;

											strcpy(pEventPipeInstance->FileDevice, "CompactFlash");
											strcpy(pEventPipeInstance->FileName, "Pipe_Type");
											ultoa(type, &pEventPipeInstance->FileName[strlen(pEventPipeInstance->FileName)]);
											strcat(pEventPipeInstance->FileName, "_Inst");
											ultoa(instance, &pEventPipeInstance->FileName[strlen(pEventPipeInstance->FileName)]);
											strcat(pEventPipeInstance->FileName, ".dat");

											pEventPipeInstance->fileOffsetWrite = 0;
											pEventPipeInstance->GetEventsFromReadPipe = TRUE;

											pEventPipeInstance->fileStep = 1;
										}
									}
									break;

								/* ----------- */
								/* File öffnen */
								/* ----------- */
								case 1:
									pEventPipeInstance->iFileOpen.enable = 1;
									pEventPipeInstance->iFileOpen.pDevice = (unsigned long)pEventPipeInstance->FileDevice;
									pEventPipeInstance->iFileOpen.pFile   = (unsigned long)pEventPipeInstance->FileName;
									pEventPipeInstance->iFileOpen.mode = FILE_RW;
									FileOpen(&pEventPipeInstance->iFileOpen);
									pEventPipeInstance->fileIdent = pEventPipeInstance->iFileOpen.ident;
									pEventPipeInstance->fileLen = pEventPipeInstance->iFileOpen.filelen;
									if (pEventPipeInstance->iFileOpen.status == fiERR_FILE_NOT_FOUND) {
										pEventPipeInstance->fileStep = 2;
									}
									else if (pEventPipeInstance->iFileOpen.status == 0) {
										pEventPipeInstance->fileStep = 3;
									}
									else if (pEventPipeInstance->iFileOpen.status != 65535) {
										pEventPipeInstance->fileState = pEventPipeInstance->iFileOpen.status;
										pEventPipeInstance->fileStep = 8;
									}
									break;

								/* ------------ */
								/* File anlegen */
								/* ------------ */
								case 2:
									pEventPipeInstance->iFileCreate.enable = 1;
									pEventPipeInstance->iFileCreate.pDevice = (unsigned long)pEventPipeInstance->FileDevice;
									pEventPipeInstance->iFileCreate.pFile   = (unsigned long)pEventPipeInstance->FileName;
									FileCreate(&pEventPipeInstance->iFileCreate);
									pEventPipeInstance->fileIdent = pEventPipeInstance->iFileCreate.ident;
									if (pEventPipeInstance->iFileCreate.status == 0) {
										pEventPipeInstance->fileStep = 3;
									}
									else if (pEventPipeInstance->iFileCreate.status != 65535) {
										pEventPipeInstance->fileState = pEventPipeInstance->iFileCreate.status;
										pEventPipeInstance->fileStep = 8;
									}
									break;

								/* -------------- */
								/* File schreiben */
								/* -------------- */
								case 3:
									if (pEventPipeInstance->iFileRead.status == 0)
									{
										pEventPipeInstance->iFileWrite.enable = 1;
										pEventPipeInstance->iFileWrite.ident = pEventPipeInstance->fileIdent;
										pEventPipeInstance->iFileWrite.offset = pEventPipeInstance->fileOffsetWrite;
										pEventPipeInstance->iFileWrite.pSrc = (unsigned long)pEventPipeHeaderWrite;
										pEventPipeInstance->iFileWrite.len = sizeof(EVENT_PIPE_HEADER) + pEventPipeHeaderWrite->pipe_size;
										FileWrite(&pEventPipeInstance->iFileWrite);
										if (pEventPipeInstance->iFileWrite.status == 0) {
											pEventPipeHeaderWrite->iPipeRead = pEventPipeHeaderWrite->iPipeWrite;
											pEventPipeInstance->WriteDataBusy = FALSE;
											switch (pAccessEventPipe->ModeFileBuffer) {
												/* bis Puffergrösse */
												case 0:
													if (pEventPipeInstance->fileOffsetWrite +  sizeof(EVENT_PIPE_HEADER) + pEventPipeHeaderWrite->pipe_size < pAccessEventPipe->SizeFileBuffer) {
														pEventPipeInstance->fileOffsetWrite += sizeof(EVENT_PIPE_HEADER) + pEventPipeHeaderWrite->pipe_size;
													}
													break;
												/* Ringpuffer */
												case 1:
													if (pEventPipeInstance->fileOffsetWrite +  sizeof(EVENT_PIPE_HEADER) + pEventPipeHeaderWrite->pipe_size < pAccessEventPipe->SizeFileBuffer) {
														pEventPipeInstance->fileOffsetWrite += sizeof(EVENT_PIPE_HEADER) + pEventPipeHeaderWrite->pipe_size;
													}
													else {
														pEventPipeInstance->fileOffsetWrite = 0;
													}
													break;
												/* unendlich */
												case 2:
													pEventPipeInstance->fileOffsetWrite += sizeof(EVENT_PIPE_HEADER) + pEventPipeHeaderWrite->pipe_size;
													break;
											}
											pEventPipeInstance->BufferFileIndex = (pEventPipeInstance->BufferFileIndex + 1) % 2;
											pEventPipeInstance->fileStep = 4;
										}
										else if (pEventPipeInstance->iFileWrite.status != 65535) {
											pEventPipeInstance->WriteDataBusy = FALSE;
											pEventPipeInstance->fileState = pEventPipeInstance->iFileWrite.status;
											pEventPipeInstance->fileStep = 8;
										}
										else {
											pEventPipeInstance->WriteDataBusy = TRUE;
										}
									}
									break;

								/* --------------------- */
								/* Auf neue Daten warten */
								/* --------------------- */
								case 4:
									if (pEventPipeInstance->BufferEventIndex != pEventPipeInstance->BufferFileIndex) {
										pEventPipeInstance->fileStep = 3;
									}
									break;

								/* ----------- */
								/* File Fehler */
								/* ----------- */
								case 8:
									pEventPipeInstance->fileSysError = FileIoGetSysError();
									pEventPipeInstance->ReadDataBusy = FALSE;
									pEventPipeInstance->fileIdent = NULL;
									pEventPipeInstance->fileState = 0;
									pEventPipeInstance->fileStep = 0;
									break;

							} /* (*pfileStep) */

							/* ------------ */
							/* File - Lesen */
							/* ------------ */
							switch (pEventPipeInstance->fileStep) {

								/* ---------- */
								/* File lesen */
								/* ---------- */
								case 3:
								case 4:
									if (
										pEventPipeInstance->iFileWrite.status == 0
										&&
										(
											(
												pEventPipeHeaderRead->iPipeRead == pEventPipeHeaderRead->iPipeWrite &&
												pEventPipeInstance->fileOffsetWrite >= sizeof(EVENT_PIPE_HEADER) + pEventPipeHeaderRead->pipe_size
											)
											||
											pEventPipeInstance->ReadDataBusy == TRUE
										)
									) {
										pEventPipeInstance->iFileRead.enable = 1;
										pEventPipeInstance->iFileRead.ident = pEventPipeInstance->fileIdent;
										pEventPipeInstance->iFileRead.offset = pEventPipeInstance->fileOffsetRead;
										pEventPipeInstance->iFileRead.pDest = (unsigned long)pEventPipeHeaderRead;
										pEventPipeInstance->iFileRead.len = sizeof(EVENT_PIPE_HEADER) + pEventPipeHeaderRead->pipe_size;
										FileRead(&pEventPipeInstance->iFileRead);
										if (pEventPipeInstance->iFileRead.status == 0) {
											/* Pointer relozieren */
											pEventPipeHeaderRead->pPipeData = (unsigned char*)&pEventPipeHeaderRead[1];
											pEventPipeInstance->ReadDataBusy = FALSE;
											pEventPipeInstance->fileOffsetRead += sizeof(EVENT_PIPE_HEADER) + pEventPipeHeaderRead->pipe_size;
											if (pEventPipeInstance->fileOffsetRead >= pEventPipeInstance->fileOffsetWrite) {
												pEventPipeInstance->fileOffsetRead  = 0;
												pEventPipeInstance->fileOffsetWrite = 0;
												pEventPipeInstance->fileStep = 6;
											}
										}
										else if (pEventPipeInstance->iFileRead.status != 65535) {
											pEventPipeInstance->ReadDataBusy = FALSE;
											pEventPipeInstance->fileState = pEventPipeInstance->iFileRead.status;
											pEventPipeInstance->fileStep = 8;
										}
										else {
											pEventPipeInstance->ReadDataBusy = TRUE;
										}
									}
									else {
										#warning ! ??? !
										pEventPipeInstance->ReadDataBusy = FALSE;
									}
									break;

								/* -------------- */
								/* File schließen */
								/* -------------- */
								case 6:
									pEventPipeInstance->iFileClose.enable = 1;
									pEventPipeInstance->iFileClose.ident = pEventPipeInstance->fileIdent;
									FileClose(&pEventPipeInstance->iFileClose);
									if (pEventPipeInstance->iFileClose.status == 0) {
										pEventPipeInstance->fileStep = 7;
									}
									else if (pEventPipeInstance->iFileClose.status != 65535) {
										pEventPipeInstance->fileState = pEventPipeInstance->iFileClose.status;
										pEventPipeInstance->fileStep = 8;
									}
									break;

								/* ------------ */
								/* File löschen */
								/* ------------ */
								case 7:
									pEventPipeInstance->iFileDelete.enable = 1;
									pEventPipeInstance->iFileDelete.pDevice = (unsigned long)pEventPipeInstance->FileDevice;
									pEventPipeInstance->iFileDelete.pName = (unsigned long)pEventPipeInstance->FileName;
									FileDelete(&pEventPipeInstance->iFileDelete);
									if (pEventPipeInstance->iFileDelete.status == 0) {
										pEventPipeInstance->WriteDataBusy = FALSE;
										pEventPipeInstance->ReadDataBusy = FALSE;
										pEventPipeInstance->fileIdent = NULL;
										pEventPipeInstance->fileState = 0;
										pEventPipeInstance->fileStep = 0;
									}
									else if (pEventPipeInstance->iFileDelete.status != 65535) {
										pEventPipeInstance->fileState = pEventPipeInstance->iFileDelete.status;
										pEventPipeInstance->fileStep = 8;
									}
									break;

								/* ----------- */
								/* File Fehler */
								/* ----------- */
								case 8:
									pEventPipeInstance->fileSysError = FileIoGetSysError();
									pEventPipeInstance->WriteDataBusy = FALSE;
									pEventPipeInstance->ReadDataBusy = FALSE;
									pEventPipeInstance->fileIdent = NULL;
									pEventPipeInstance->fileState = 0;
									pEventPipeInstance->fileStep = 0;
									break;

							} /* (*pfileStep) */
						} /* (pEventPipeHeaderWrite != NULL && pEventPipeHeaderRead != NULL) */
					} /* (pEventPipeInstance->WriteToFile == TRUE) */
				} /* (pAccessEventPipe != NULL) */
			} /* (type = 0; type < pAccessServer->countType; type++) */
		} /* (instance = 0; instance < pAccessServer->countEventInstance; instance++) */
		return 0;
	} /* (idBrServer != NULL) */
	else {
		return cEC_INVALID_SERVER;
	}
} /* CopyPipeToFile */

/*============================= Ende der Datei ==============================*/
```
